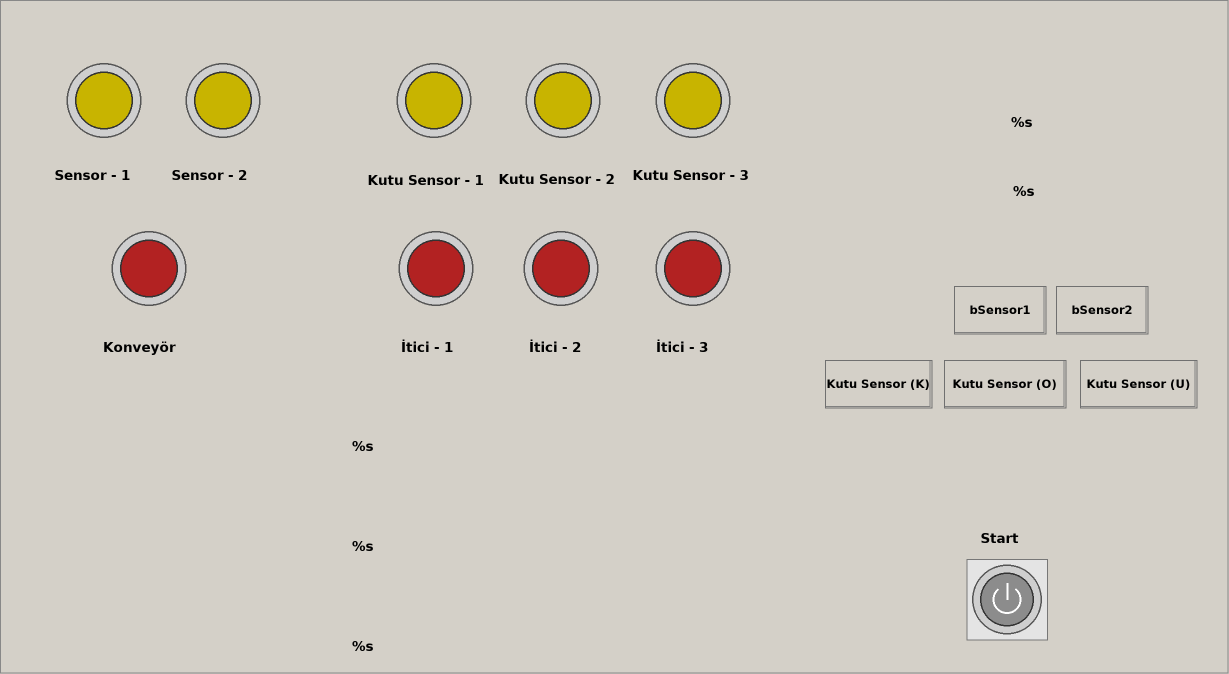
VISUALIZATION VISU_1  // 1229x674
    PowerSwitch (964,559 86x81), variable: MAIN.bButon, behaviour: TOGGLE, style: Switch-PowerSwitch-Gray
    Button (954,286 92x48), "bSensor1"
        toggle MAIN.bSensor1
    Button (1056,286 92x48), "bSensor2"
        toggle MAIN.bSensor2
    Label (951,511 97x55), "Start"
    Button (825,360 107x48), "Kutu Sensor (K)"
        toggle MAIN.bKutuSens1
    Button (944,360 122x48), "Kutu Sensor (O)"
        toggle MAIN.bKutuSens2
    Button (1080,360 117x48), "Kutu Sensor (U)"
        toggle MAIN.bKutuSens3
    Lamp1 (52,57 104x87), variable: MAIN.bSensor1, style: Lamp-Lamp1-Yellow
    Lamp1 (171,57 104x87), variable: MAIN.bSensor2, style: Lamp-Lamp1-Yellow
    Lamp1 (382,57 104x87), variable: MAIN.bKutuSens1, style: Lamp-Lamp1-Yellow
    Lamp1 (511,57 104x87), variable: MAIN.bKutuSens2, style: Lamp-Lamp1-Yellow
    Lamp1 (641,57 104x87), variable: MAIN.bKutuSens3, style: Lamp-Lamp1-Yellow
    Lamp1 (97,225 104x87), variable: MAIN.bHat, style: Lamp-Lamp1-Red
    Lamp1 (384,225 104x87), variable: MAIN.bKol1, style: Lamp-Lamp1-Red
    Lamp1 (509,225 104x87), variable: MAIN.bKol2, style: Lamp-Lamp1-Red
    Lamp1 (641,225 104x87), variable: MAIN.bKol3, style: Lamp-Lamp1-Red
    Rectangle (105,419 516x55), "%s", text variable: MAIN.sMsgKisa_1
    Rectangle (105,519 516x55), "%s", text variable: MAIN.sMsgOrta_1
    Rectangle (105,619 516x55), "%s", text variable: MAIN.sMsgUzun_1
    Label (91,320 97x55), "Konveyör"
    Label (379,320 97x55), "İtici - 1"
    Label (507,320 97x55), "İtici - 2"
    Label (634,320 97x55), "İtici - 3"
    Label (44,148 97x55), "Sensor - 1"
    Label (161,148 97x55), "Sensor - 2"
    Label (357,153 142x55), "Kutu Sensor - 1"
    Label (486,152 142x55), "Kutu Sensor - 2"
    Label (620,148 142x55), "Kutu Sensor - 3"
    Rectangle (817,95 410x55), "%s", text variable: MAIN.sInfoMsg
    Rectangle (819,164 410x55), "%s", text variable: MAIN.sMsgYukseklik
END_VISUALIZATION

(* stored: Version 1.1.0.1, ProductVersion 3.1.4024.4
   Visu VISU_1: Id {40db4f35-4822-4a90-8567-2335099c9071} *)
